// TIA Portal V17 export
// export: Created 2025-06-26T06:49:12.4434232Z, ExportSetting WithDefaults, DisplayName Totally Integrated Automation Portal, DisplayVersion V17 Update 8, DisplayName TIA Portal Openness, DisplayVersion V17 Update 8, DisplayName TIA Portal Version Control Interface, DisplayVersion V17, DisplayName STEP 7 Professional, DisplayVersion V17 Update 8, DisplayName STEP 7 Safety, DisplayVersion V17 Update 6, DisplayName WinCC Advanced, DisplayVersion V17 Update 8
FUNCTION_BLOCK "PerformanceControl"   // FB9, FBD
TITLE = Performance control
{ S7_Optimized_Access := 'TRUE' }
VERSION : 0.1
// POWER Restiction IDs:
//   1: Customer: Heat sink suction temperature
//   2: Customer: Heat source discharge temperature
//   3: Customer: Heat sink discharge temperature
//   4: Customer: Heat source suction temperature
//   5: Customer: Reserve Analog In
//   6: Customer: Variable control
//   7: Customer: Reserve
//   8: Safety: Safety limit condensing pressure
//   9: Safety: Safety limit compressor motor torque
// 10: Safety: Safety limit compressor motor winding temperature
// 11: Safety: Safety limit container air temperature
// 12: Safety: Safety limit control cabinet air temperature
// 13: Safety: Safety limit compressor inverter temperature
// 14: Safety: Safety limit oil sump oil temperature
// stored: AutoNumber true, IsIECCheckEnabled false, IsRetainMemResEnabled false, MemoryReserve 100, SetENOAutomatically false, UDAEnableTagReadback false
   VAR_INPUT
      bReset { ExternalAccessible := 'False'; ExternalVisible := 'False'; ExternalWritable := 'False'} : Bool;
   END_VAR
   VAR_OUTPUT
      T_AddSuperheat_Controlled { ExternalAccessible := 'False'; ExternalVisible := 'False'; ExternalWritable := 'False'} : Real;
      CompressorPerformanceSetpoint { ExternalAccessible := 'False'; ExternalVisible := 'False'; ExternalWritable := 'False'} : Real;
      RunningCondition { ExternalAccessible := 'False'; ExternalVisible := 'False'; ExternalWritable := 'False'} : Bool;
      RestrictionID { ExternalAccessible := 'False'; ExternalVisible := 'False'; ExternalWritable := 'False'} : Int;
      TargetValue { ExternalAccessible := 'False'; ExternalVisible := 'False'; ExternalWritable := 'False'} : Real;
      CurrentValue { ExternalAccessible := 'False'; ExternalVisible := 'False'; ExternalWritable := 'False'} : Real;
      Rate { ExternalAccessible := 'False'; ExternalVisible := 'False'; ExternalWritable := 'False'} : Real;
   END_VAR
   VAR
      PerformanceRate { ExternalAccessible := 'False'; ExternalVisible := 'False'; ExternalWritable := 'False'} : Real;
      LastDT1_Memory_n { ExternalAccessible := 'False'; ExternalVisible := 'False'; ExternalWritable := 'False'} : Real;
      IntegralPart_Memory_n { ExternalAccessible := 'False'; ExternalVisible := 'False'; ExternalWritable := 'False'} : Real;
      ParameterChange_Memory_n { ExternalAccessible := 'False'; ExternalVisible := 'False'; ExternalWritable := 'False'} : Real;
      LowerSpeedLimit_Reached { ExternalAccessible := 'False'; ExternalVisible := 'False'; ExternalWritable := 'False'} : Bool;
      UpperSpeedLimit_Reached { ExternalAccessible := 'False'; ExternalVisible := 'False'; ExternalWritable := 'False'} : Bool;
      PowerTimer { ExternalAccessible := 'False'; ExternalVisible := 'False'; ExternalWritable := 'False'; S7_SetPoint := 'True'} : IEC_TIMER;
      HeatSinkTimer { ExternalAccessible := 'False'; ExternalVisible := 'False'; ExternalWritable := 'False'; S7_SetPoint := 'True'} : IEC_TIMER;
      HeatSourceTimer { ExternalAccessible := 'False'; ExternalVisible := 'False'; ExternalWritable := 'False'; S7_SetPoint := 'True'} : IEC_TIMER;
      VariableControlTimer { ExternalAccessible := 'False'; ExternalVisible := 'False'; ExternalWritable := 'False'; S7_SetPoint := 'True'} : IEC_TIMER;
      EngineRequired { ExternalAccessible := 'False'; ExternalVisible := 'False'; ExternalWritable := 'False'} : Bool := true;
      DT1_storage { ExternalAccessible := 'False'; ExternalVisible := 'False'; ExternalWritable := 'False'} : Real;
   END_VAR
   VAR_TEMP
      Dummy : Real;
      Target : Struct
         ID : Int;
         Error : Real;
         Target : Real;
         CurrentValue : Real;
         Kp : Real;
         Tn : Int;
         Tv : Int;
      END_STRUCT;
      T_Setpoint : Real;
      T_CurrentValue : Real;
      ManualControl_acv : Bool;
      DT_Source : Real;
      DT_Sink : Real;
      DT_VarCont : Real;
      ID : USInt;
      AddPressSafetyMargin : Real;
      ControlError : Real;
   END_VAR
   VAR CONSTANT
      KP_STEMP : Real := 20.0;
      TN_STEMP : Int := 120;
      i0 : Int := 0;
   END_VAR
BEGIN

REGION Network 1: Reset manual modes
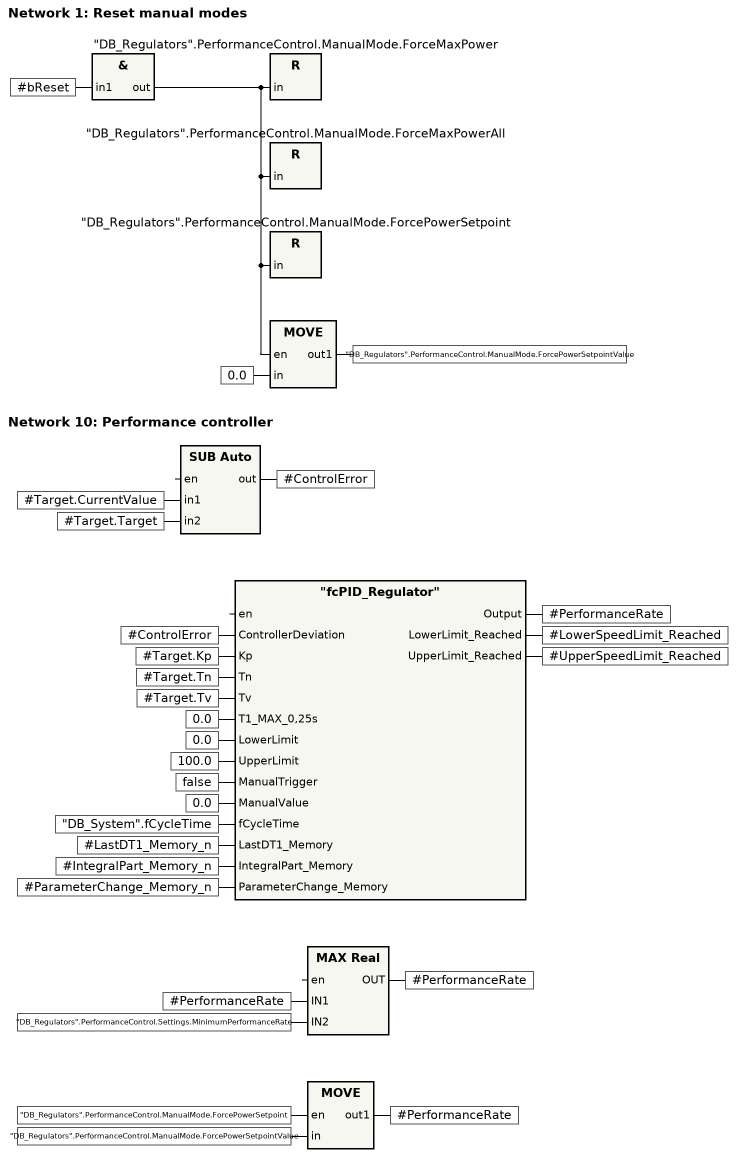
   IF #bReset THEN
       "DB_Regulators".PerformanceControl.ManualMode.ForceMaxPower := FALSE;
       "DB_Regulators".PerformanceControl.ManualMode.ForceMaxPowerAll := FALSE;
       "DB_Regulators".PerformanceControl.ManualMode.ForcePowerSetpoint := FALSE;
       "DB_Regulators".PerformanceControl.ManualMode.ForcePowerSetpointValue := 0.0;
   END_IF;
END_REGION

REGION Network 2 (SCL): Preset
   #ManualControl_acv := "DB_Regulators".PerformanceControl.ManualMode.ForceMaxPower OR "DB_Regulators".PerformanceControl.ManualMode.ForceMaxPowerAll OR "DB_Regulators".PerformanceControl.ManualMode.ForcePowerSetpoint;

   // Preset
   #Target.Tv := 0;
   #Target.Error := 20; // Positive value between 0.1-100, larger values mean the controller intervenes longer before the setpoint is reached, if it changes rapidly.
   #Target.Tn := REAL_TO_INT(#Target.Error * "DB_Regulators".PerformanceControl.Settings.Config.INCREASEWITHNORESTRICTION); // 
   #Target.Kp := 1;
END_REGION

REGION Network 3 (SCL): Heat sink control (Restrictions 1 & 2)
    IF "DB_Regulators".PerformanceControl.Settings.HeatSink.Control_Active THEN
      #T_Setpoint := "DB_Regulators".PerformanceControl.Settings.HeatSink.Setpoint;

       // NOTE! Feed Flow here means "discharge"
      IF "DB_Regulators".PerformanceControl.Settings.HeatSink.UseFeedFlow THEN
           // Heat sink discharge temperature
           #T_CurrentValue := "DB_AI".HBL_TT_518.Eng.fValue;
           #ID := USInt#2;
       ELSE
           // Heat sink suction temperature
           #T_CurrentValue := "DB_AI".HBL_TT_901.Eng.fValue;
           #ID := USInt#1;
       END_IF;
       #DT_Sink := #T_CurrentValue - #T_Setpoint;

       "Restriction"(ID := #ID,
                     Target := #T_Setpoint,
                     Value := #T_CurrentValue,
                     Kp := "DB_Regulators".PerformanceControl.Settings.HeatSink.Kp,
                     Tn := REAL_TO_INT("DB_Regulators".PerformanceControl.Settings.HeatSink.Tn),
                     Tv := #i0,
                     fCycleTime:= "DB_System".fCycleTime,
                     IO := #Target,
                     DT1_storage := #Dummy);
   END_IF;
END_REGION

REGION Network 4 (SCL): Heat source control (Restrictions 3 & 4)
    IF "DB_Regulators".PerformanceControl.Settings.HeatSource.Control_Active THEN
       #T_Setpoint := "DB_Regulators".PerformanceControl.Settings.HeatSource.Setpoint;

       // NOTE! "Feed flow" here means "suction"
       IF "DB_Regulators".PerformanceControl.Settings.HeatSource.UseFeedFlow THEN
           // Heat source suction temperature
           #T_CurrentValue := "DB_AI".HBL_TT_546.Eng.fValue;
           #ID := USInt#4;
       ELSE
           // Heat source discharge temperature
           #T_CurrentValue := "DB_AI".HBL_TT_542.Eng.fValue;
           #ID := USInt#3;

       END_IF;
       #DT_Source := #T_Setpoint - #T_CurrentValue;

       "Restriction"(ID := #ID,
                     Target := #T_Setpoint,
                     Value := #T_CurrentValue,
                     Kp := "DB_Regulators".PerformanceControl.Settings.HeatSource.Kp,
                     Tn := REAL_TO_INT("DB_Regulators".PerformanceControl.Settings.HeatSource.Tn),
                     Tv := #i0,
                     fCycleTime := "DB_System".fCycleTime,
                     IO := #Target,
                     DT1_storage := #Dummy);
   END_IF;
END_REGION

REGION Network 5 (SCL): Variable control (Restriction 6)
   IF "DB_Regulators".PerformanceControl.Settings.VariableControl.Control_Active AND "DB_Regulators".PerformanceControl.Settings.VariableControl.ReferenceID > 0 THEN
       #T_Setpoint := "DB_Regulators".PerformanceControl.Settings.VariableControl.Setpoint;

       CASE "DB_Regulators".PerformanceControl.Settings.VariableControl.ReferenceID OF
           1:
               #T_CurrentValue := "DB_AI".HBL_TT_901.Eng.fValue;
           2:
               #T_CurrentValue := "DB_AI".HBL_TT_518.Eng.fValue;
           3:
               #T_CurrentValue := "DB_Calc".HeatSink.DeltaT.fValue;
           4:
               #T_CurrentValue := "DB_AI".HBL_TT_542.Eng.fValue;
           5:
               #T_CurrentValue := "DB_AI".HBL_TT_546.Eng.fValue;
           6:
               #T_CurrentValue := "DB_Calc".HeatSource.DeltaT.fValue;
           7:
               #T_CurrentValue := 0; //Extern Temperature Sensor
           ELSE  // Statement section ELSE
               #T_CurrentValue := 0;
       END_CASE;
       #DT_VarCont := #T_CurrentValue - #T_Setpoint;

       "Restriction"(ID := 6,
                     Target := #T_Setpoint,
                     Value := #T_CurrentValue,
                     Kp := "DB_Regulators".PerformanceControl.Settings.VariableControl.Kp,
                     Tn := REAL_TO_INT("DB_Regulators".PerformanceControl.Settings.VariableControl.Tn),
                     Tv := #i0,
                     fCycleTime := "DB_System".fCycleTime,
                     IO := #Target,
                     DT1_storage := #Dummy);
   END_IF;
END_REGION

REGION Network 6 (SCL): Safety limit condensing pressure (Restriction 8)
   // If condensing temperature is close or above Heat sink feed temperature, increase safety margin  (-2K - 4K) difference   => (0 - 300kPa) extra
   #AddPressSafetyMargin := LIMIT_REAL(IN := ("DB_Calc".HighPressPart.CondenserSaturationTemperature.fValue - "DB_AI".HBL_TT_518.Eng.fValue + 2) * 50, MN := 0, MX := 300);

   // If condensing maximum pressure is close or above critical point, increase safety margin         (0 - 400kPa) difference => (0 - 200kPa) extra
   #AddPressSafetyMargin += LIMIT_REAL(IN := ("DB_CurrentSetting".System.Limits.p_CompressorOut_Max - "DB_CurrentSetting".Fluid.P_CriticalPoint) * 0.5, MN := 0, MX := 200);

   "Restriction"(ID:=8,
                 Target:="DB_CurrentSetting".System.Limits.p_CompressorOut_Max - 200.0 - #AddPressSafetyMargin,
                 Value:="DB_AI".HBL_PT_517.Eng.fValue,
                 Kp:=0.36,
                 Tn:=16,
                 Tv:=25,
                 fCycleTime := "DB_System".fCycleTime,
                 IO:=#Target,
                 DT1_storage:=#DT1_storage);
END_REGION

REGION Network 7 (SCL): Safety limit torque (Restriction 9)
   // ##REVIEW THIS!! Should be operating at 100% torque limit unless some good reason for it?
   // Safety limit compressor motor torque (110Nm @ 1500rpm)
   "Restriction"(ID:=9,
                 Target:=110.0*SQRT(1500/"DB_InverterDrives".HBL_SC_10.Stat.Speed.Eng.fValue),
                 Value:= "DB_InverterDrives".HBL_SC_10.Stat.Torque.Eng.fValue,
                 Kp:=0.04,
                 Tn:=3,
                 Tv:=#i0,
                 fCycleTime:= "DB_System".fCycleTime,
                 IO:=#Target,
                 DT1_storage:=#Dummy);
END_REGION

REGION Network 8 (SCL): Safety limit temperatures (Restriction 10, 11, 12, 14)
    // Safety limit compressor motor winding temperature
   "Restriction"(ID:=10,
                 Target:="DB_CurrentSetting".Compressor.Limits.T_Motor_Max - 5,
                 Value:="DB_AI".HBL_TT_20.Eng.fValue,
                 Kp:=#KP_STEMP,
                 Tn:=#TN_STEMP,
                 Tv:=#i0,
                 fCycleTime := "DB_System".fCycleTime,
                 IO:=#Target,
                 DT1_storage:=#Dummy);
   // Safety limit container air temperature
   "Restriction"(ID:=11,
                 Target:="DB_CurrentSetting".System.Limits.T_Housing_Max - 5,
                 Value:="DB_AI".HBL_TT_16.Eng.fValue,
                 Kp:=#KP_STEMP,
                 Tn:=#TN_STEMP,
                 Tv:=#i0,
                 fCycleTime := "DB_System".fCycleTime,
                 IO:=#Target,
                 DT1_storage:=#Dummy);
   // Safety limit control cabinet air temperature
   "Restriction"(ID:=12,
                 Target:="DB_CurrentSetting".StaticSetting.Limits.T_Cabinet_Max - 3,
                 Value:="DB_AI".HBL_TT_17.Eng.fValue,
                 Kp:=#KP_STEMP,
                 Tn:=#TN_STEMP,
                 Tv:=#i0,
                 fCycleTime := "DB_System".fCycleTime,
                 IO:=#Target,
                 DT1_storage:=#Dummy);
   // Safety limit compressor inverter temperature
   (*
   "Restriction"(ID:=13,
                 Target:="DB_CurrentSetting".CompressorTypes.Limits.T_Inverter_Max - 5,
                 Value:="DB_SensorInputs".Compressors.T19_Inverter,
                 Kp:=#KP_STEMP,
                 Tn:=#TN_STEMP,
                 Tv:=#i0,
                 fCycleTime:= "DB_System".fCycleTime,
                 IO:=#Target,
                 DT1_storage:=#Dummy);
   *)
   // Safety limit oil sump oil temperature (Max - 5°C)
   "Restriction"(ID:=14,
                 Target:="DB_CurrentSetting".Fluid.Limits.T_OilTemperature_Critical - 5,
                 Value:="DB_AI".HBL_TT_03.Eng.fValue,
                 Kp:=#KP_STEMP,
                 Tn:=#TN_STEMP,
                 Tv:=#i0,
                 fCycleTime := "DB_System".fCycleTime,
                 IO:=#Target,
                 DT1_storage:=#Dummy);
END_REGION

REGION Network 9 (SCL): Force max power
   // Bypass all power limitations. Self-protection limitations included
   IF "DB_Regulators".PerformanceControl.ManualMode.ForceMaxPowerAll THEN
       #Target.Error := 10.0;
       #Target.ID := 0;
       #Target.Kp  := #KP_STEMP;
       #Target.Tn  := #TN_STEMP;
   END_IF;
END_REGION

REGION Network 10: Performance controller
   // ###NOTSURE disable the manual mode (overwrites output instead in FB34)
   #ControlError := #Target.CurrentValue - #Target.Target;
   "fcPID_Regulator"(ControllerDeviation := #ControlError,
                     Kp := #Target.Kp,
                     Tn := #Target.Tn,
                     Tv := #Target.Tv,
                     "T1_MAX_0,25s" := 0.0,
                     LowerLimit := 0.0,
                     UpperLimit := 100.0,
                     ManualTrigger := false,
                     ManualValue := 0.0,
                     fCycleTime := "DB_System".fCycleTime,
                     LastDT1_Memory := #LastDT1_Memory_n,
                     IntegralPart_Memory := #IntegralPart_Memory_n,
                     ParameterChange_Memory := #ParameterChange_Memory_n,
                     Output => #PerformanceRate,
                     LowerLimit_Reached => #LowerSpeedLimit_Reached,
                     UpperLimit_Reached => #UpperSpeedLimit_Reached);
   #PerformanceRate := MAX(IN1 := #PerformanceRate, IN2 := "DB_Regulators".PerformanceControl.Settings.MinimumPerformanceRate);
   IF "DB_Regulators".PerformanceControl.ManualMode.ForcePowerSetpoint THEN
       #PerformanceRate := "DB_Regulators".PerformanceControl.ManualMode.ForcePowerSetpointValue;
   END_IF;
END_REGION

REGION Network 11 (SCL): Outputs
   //If there is no nagative restriction and the Powersetpoint is 100%. Don't show restrictions.
   IF #Target.Error > 0 AND #PerformanceRate >= 98 THEN 
       #Target.ID := 0;
   END_IF;

   // Local outputs
   IF #EngineRequired AND ("DB_State".State."5_Warmup" OR "DB_State".State."6_Running") THEN
       #Rate := #PerformanceRate;
   ELSE
       #Rate := 0;
   END_IF;

   "DB_Regulators".PerformanceControl.RestrictionID := #RestrictionID := #Target.ID;
   "DB_Regulators".PerformanceControl.TargetValue := #TargetValue := #Target.Target;
   "DB_Regulators".PerformanceControl.CurrentValue := #CurrentValue := #Target.CurrentValue;
   "DB_Regulators".PerformanceControl.fOut := #CompressorPerformanceSetpoint := #PerformanceRate;
END_REGION

REGION Network 12 (SCL): AdditionalSuperheatRequest
   // If the performance rate is below a minimum (X%) an additional superheat is required. The maximum required superheat (UpperAdditionalSuperheatLimit) is reached if the power requirement is 0;
   // Ab einer Leistung kleiner X% soll ein zusätzliches Superheat angefordert werden. Maximal MaximumAdditionalSuperheat
   #T_AddSuperheat_Controlled := MAX(IN1:= ("DB_Regulators".PerformanceControl.Settings.Config.MinimumPerformanceRequirement-#PerformanceRate)/"DB_Regulators".PerformanceControl.Settings.Config.MinimumPerformanceRequirement, 
                                     IN2:= 0)*"DB_Regulators".PerformanceControl.Settings.Config.MaximumAdditionalSuperheat;
END_REGION

REGION Network 13 (SCL): Validate standby/operational limits
   // Validate settings
   IF "DB_Regulators".PerformanceControl.Settings.HeatSink.DT_Limit_Standby < - "DB_Regulators".PerformanceControl.Settings.HeatSink.DT_Limit_Resume THEN
       "DB_Regulators".PerformanceControl.Settings.HeatSink.DT_Limit_Resume := "DB_Regulators".PerformanceControl.Settings.HeatSink.DT_Limit_Standby;
   END_IF;
   IF "DB_Regulators".PerformanceControl.Settings.HeatSource.DT_Limit_Standby < - "DB_Regulators".PerformanceControl.Settings.HeatSource.DT_Limit_Resume THEN
       "DB_Regulators".PerformanceControl.Settings.HeatSource.DT_Limit_Resume := "DB_Regulators".PerformanceControl.Settings.HeatSource.DT_Limit_Standby;
   END_IF;
   IF "DB_Regulators".PerformanceControl.Settings.VariableControl.DT_Limit_Standby < - "DB_Regulators".PerformanceControl.Settings.VariableControl.DT_Limit_Resume THEN
       "DB_Regulators".PerformanceControl.Settings.VariableControl.DT_Limit_Resume := "DB_Regulators".PerformanceControl.Settings.VariableControl.DT_Limit_Standby;
   END_IF;
END_REGION

REGION Network 14 (SCL): Running condition
   // 

   IF #EngineRequired THEN
       // Running condition is true, see if we need to reset it
       #PowerTimer.TON(IN:=("DB_Regulators".PerformanceControl.Settings.SwitchToStandby_timeDelay <> T#0s) AND 
                           (#PerformanceRate <= "DB_Regulators".PerformanceControl.Settings.MinimumPerformanceRate), PT := "DB_Regulators".PerformanceControl.Settings.SwitchToStandby_timeDelay + T#1ms);

       #HeatSinkTimer.TON(IN:= "DB_Regulators".PerformanceControl.Settings.HeatSink.Control_Active AND 
                               (#DT_Sink >= "DB_Regulators".PerformanceControl.Settings.HeatSink.DT_Limit_Standby), PT:= T#1s);
       #HeatSourceTimer.TON(IN:= "DB_Regulators".PerformanceControl.Settings.HeatSource.Control_Active AND 
                                (#DT_Source >= "DB_Regulators".PerformanceControl.Settings.HeatSource.DT_Limit_Standby), PT:= T#1s);
       #VariableControlTimer.TON(IN := "DB_Regulators".PerformanceControl.Settings.VariableControl.Control_Active AND 
                                       (#DT_VarCont >= "DB_Regulators".PerformanceControl.Settings.VariableControl.DT_Limit_Standby), PT := T#1s);
       IF (#PowerTimer.Q OR #HeatSinkTimer.Q OR #HeatSourceTimer.Q OR #VariableControlTimer.Q) AND NOT #ManualControl_acv THEN
           PRESET_TIMER("TIMER":=#PowerTimer,PT:=T#1ms);
           PRESET_TIMER("TIMER":=#HeatSinkTimer,PT:=T#1ms);    
           PRESET_TIMER("TIMER":=#HeatSourceTimer,PT:=T#1ms);
           PRESET_TIMER("TIMER" := #VariableControlTimer,PT := T#1ms);
           #EngineRequired := false;
       END_IF;
   ELSE
       // Running condition is false, see if we need to set it
       #PowerTimer.TOF(IN:=("DB_Regulators".PerformanceControl.Settings.SwitchToStandby_timeDelay <> T#0s) AND 
                           (#PerformanceRate <= "DB_Regulators".PerformanceControl.Settings.MinimumPerformanceRate), PT := "DB_Regulators".PerformanceControl.Settings.SwitchToStandby_timeDelay + T#1ms);
       #HeatSinkTimer.TOF(IN:="DB_Regulators".PerformanceControl.Settings.HeatSink.Control_Active AND 
                              (#DT_Sink > - "DB_Regulators".PerformanceControl.Settings.HeatSink.DT_Limit_Resume), PT:= T#1s);
       #HeatSourceTimer.TOF(IN:= "DB_Regulators".PerformanceControl.Settings.HeatSource.Control_Active AND 
                                 (#DT_Source > - "DB_Regulators".PerformanceControl.Settings.HeatSource.DT_Limit_Resume), PT:= T#1s);
       #VariableControlTimer.TOF(IN := "DB_Regulators".PerformanceControl.Settings.VariableControl.Control_Active AND 
                                       (#DT_VarCont > - "DB_Regulators".PerformanceControl.Settings.VariableControl.DT_Limit_Resume), PT := T#1s);
       IF NOT(#PowerTimer.Q OR #HeatSinkTimer.Q OR #HeatSourceTimer.Q OR #VariableControlTimer.Q) OR #ManualControl_acv THEN
           RESET_TIMER(#PowerTimer);
           RESET_TIMER(#HeatSinkTimer);
           RESET_TIMER(#HeatSourceTimer);
           RESET_TIMER(#VariableControlTimer);
           #EngineRequired := true;
       END_IF;
   END_IF;
   #RunningCondition:= #EngineRequired;
   "DB_Regulators".PerformanceControl.RunningCondition := #EngineRequired;
END_REGION
END_FUNCTION_BLOCK
